TYPE ST_PIP :
STRUCT
(* Interlock *)
   xHV_ExtIlk : BOOL; 

	rHVEna_SP : REAL := 1.0E-4;	
	
(* EPICS Controls *)	
	i_xHVEna_SW : BOOL; 
	
(* Controls *)
	q_xHVEna_DO : BOOL;	



END_STRUCT
END_TYPE

(* stored: Version 1.1.0.1, ProductVersion 3.1.4022.10
   DUT ST_PIP: Id {e391599b-61b0-45e4-858a-1c40e25414f4} *)
